TYPE ACRMemoryIntEvent EXTENDS ACRMemoryEvent :
STRUCT
	_Value : INT;
END_STRUCT
END_TYPE

(* stored: Version 1.1.0.1, ProductVersion 3.1.4020.12
   DUT ACRMemoryIntEvent: Id {e81da7c6-48a1-4d49-b2bd-526d6be55b93} *)
